(* add offset to POINTER TO WORD value *)
FUNCTION F_PointerToWordADD : PVOID
VAR_INPUT
	pPointer		: PVOID;	(* base pointer *)
	nOffset			: UDINT;			(* pointer offset *)
END_VAR
VAR
	nPointer		: ULINT;
	nPointerOffset	: ULINT;
END_VAR
(*
-------------------------------------------------------------------------------------------------
Date		Version	Author	Comments
-------------------------------------------------------------------------------------------------
30/01/2015	3.00.00	PB		No change

-------------------------------------------------------------------------------------------------
05/02/10	1.00.00	PB		Initial release

-------------------------------------------------------------------------------------------------
*)

nPointer := pPointer;					(* convert pointer to UDINT *)
nPointerOffset := nPointer + nOffset;	(* add offset *)
F_PointerToWordADD := nPointerOffset;	(* convert UDINT back to pointer *)

END_FUNCTION

(* stored: Version 1.1.0.1
   POU F_PointerToWordADD: Id {13bf8aa3-d6a4-478e-94c0-d2b099252a7b}, SpecialFunc None *)
